VAR_GLOBAL
	aBuffer:				ARRAY[0..99] OF FB_Message;
    nBuffer:				UINT := 0;
END_VAR

(* stored: Version 1.1.0.1
   GVL GVL: Id {8c417638-2928-4f7d-b718-658b035f50d1} *)
